FUNCTION F_SetAllMoversRotation : BOOL
VAR_INPUT
	Set			:ST_MoveDynamics;
END_VAR
VAR
	i			:UDINT;
END_VAR

FOR i:=1 TO XPlanar.MoverCount DO
	IF ip.Movers[i]<>0 THEN
		ip.Movers[i].Dynamics.Rotation:=Set;		
	END_IF			
END_FOR

END_FUNCTION

(* stored: Version 1.1.0.1, ProductVersion 3.1.4026.18
   POU F_SetAllMoversRotation: Id {50e85050-42e9-41cd-9929-3a6834614d12}, SpecialFunc None *)
